// TIA Portal project "ap1_2019" (V15.1)

(* hardware
DEVICE "S7300/ET200M station_1"  S7-300 station
   slot 0: "Rail_0"  Rail  6ES7 390-1***0-0AA0
   slot 2: "PLC_1"  CPU 314C-2 PN/DP  6ES7 314-6EH04-0AB0  V3.3
      slot 2: "PROFINET interface_1"  PN-IO
         slot 1: "Port_1"  Port
         slot 2: "Port_2"  Port
      slot 5: "DI 24/DO 16_1"  DI24/DO16
      slot 6: "AI 5/AO 2_1"  AI5/AO2
      slot 7: "Count_1"  Counter
      slot 8: "Positioning_1"  Positioning
   slot 4: "DO 8x24VDC/2A_1"  DO8 x 24VDC / 2A  6ES7 322-1BF01-0AA0
DEVICE "HMI_1"  KTP900 Basic PN
   slot 0: "HMI_1"  KTP900 Basic PN  6AV2 123-2JB03-0AX0  15.1.0.0
   slot 1: "HMI_RT_1"  KTP900 Basic PN  6AV2 123-2JB03-0AX0  15.1.0.0
   slot 5: "HMI_1.IE_CP_1"  PROFINET Interface  15.0.1.0
      slot 1: "PROFINET Interface_1"  PROFINET Interface
         slot 1: "Port_1"  Port
*)

// ===== PLC "PLC_1"  CPU 314C-2 PN/DP =====

VAR_GLOBAL   // PLC tag table "Default tag table"
   "F5" AT %I0.0 : Bool;
   "S3" AT %I0.1 : Bool;
   "S4" AT %I0.2 : Bool;
   "S5" AT %I0.3 : Bool;
   "S6" AT %I0.4 : Bool;
   "S7" AT %I0.5 : Bool;
   "S8" AT %I0.6 : Bool;
   "S9" AT %I0.7 : Bool;
   "S10" AT %I1.0 : Bool;
   "S11" AT %I1.1 : Bool;
   "Reserve1" AT %I1.2 : Bool;
   "BP1" AT %I1.3 : Bool;
   "B1" AT %I1.4 : Bool;
   "B2" AT %I1.5 : Bool;
   "Reserve2" AT %I1.6 : Bool;
   "B11" AT %I1.7 : Bool;
   "B12" AT %I2.0 : Bool;
   "B21" AT %I2.1 : Bool;
   "B22" AT %I2.2 : Bool;
   "B31" AT %I2.3 : Bool;
   "B32" AT %I2.4 : Bool;
   "Reserve3" AT %I2.5 : Bool;
   "Reserve4" AT %I2.6 : Bool;
   "Reserve5" AT %I2.7 : Bool;
   "M11" AT %Q0.0 : Bool;
   "M21" AT %Q0.2 : Bool;
   "M22" AT %Q0.3 : Bool;
   "M31" AT %Q0.4 : Bool;
   "M32" AT %Q0.5 : Bool;
   "Reserve6" AT %Q0.6 : Bool;
   "Reserve7" AT %Q0.7 : Bool;
   "P32" AT %Q1.0 : Bool;
   "P33" AT %Q1.1 : Bool;
   "Reserve8" AT %Q1.2 : Bool;
   "P2" AT %Q1.3 : Bool;
   "P3" AT %Q1.4 : Bool;
   "P4" AT %Q1.5 : Bool;
   "P5" AT %Q1.6 : Bool;
   "P6" AT %Q1.7 : Bool;
   "P7" AT %Q2.0 : Bool;
   "Reserve9" AT %Q2.1 : Bool;
   "P10" AT %Q2.2 : Bool;
   "P11" AT %Q2.3 : Bool;
   "P12" AT %Q2.4 : Bool;
   "P13" AT %Q2.5 : Bool;
   "P14" AT %Q2.6 : Bool;
   "P15" AT %Q2.7 : Bool;
   "M12" AT %Q0.1 : Bool;
   "MBP1" AT %M0.0 : Bool;
   "MS3" AT %M0.1 : Bool;
   "MS4" AT %M0.2 : Bool;
   "MF5" AT %M0.3 : Bool;
   "MS5" AT %M0.4 : Bool;
   "MS6" AT %M0.5 : Bool;
   "MS7" AT %M0.6 : Bool;
   "MS8" AT %M0.7 : Bool;
   "MS9" AT %M1.0 : Bool;
   "MS10" AT %M1.1 : Bool;
   "MS11" AT %M1.2 : Bool;
   "MB1" AT %M1.3 : Bool;
   "MB2" AT %M1.4 : Bool;
END_VAR

DATA_BLOCK "Master_DB"   // DB1
{ S7_Optimized_Access := 'FALSE' }
VERSION : 0.1
// stored: InstanceOfName Master
"Master"
BEGIN
END_DATA_BLOCK

DATA_BLOCK "safety_DB"   // DB2
{ S7_Optimized_Access := 'FALSE' }
VERSION : 0.1
// stored: InstanceOfName safety
"safety"
BEGIN
END_DATA_BLOCK

DATA_BLOCK "Clock_DB"   // DB5
{ S7_Optimized_Access := 'FALSE' }
VERSION : 0.1
// stored: InstanceOfName Clock
"Clock"
BEGIN
END_DATA_BLOCK

DATA_BLOCK "Indicator_DB"   // DB6
{ S7_Optimized_Access := 'FALSE' }
VERSION : 0.1
// stored: InstanceOfName Indicator
"Indicator"
BEGIN
END_DATA_BLOCK

DATA_BLOCK "Trigger_DB"   // DB7
{ S7_Optimized_Access := 'FALSE' }
VERSION : 0.1
// stored: InstanceOfName Trigger
"Trigger"
BEGIN
END_DATA_BLOCK

DATA_BLOCK "Auto_DB"   // DB9
{ S7_Optimized_Access := 'FALSE' }
VERSION : 0.1
// stored: InstanceOfName Auto
"Auto"
BEGIN
END_DATA_BLOCK

DATA_BLOCK "HMI"   // DB14
{ S7_Optimized_Access := 'FALSE' }
VERSION : 0.1
   VAR
      "Control Panel" : Bool;
   END_VAR
BEGIN
END_DATA_BLOCK

DATA_BLOCK "Total_DB"   // DB23
{ S7_Optimized_Access := 'FALSE' }
VERSION : 0.1
// stored: InstanceOfName Total
"Total"
BEGIN
END_DATA_BLOCK

FUNCTION_BLOCK "Master"   // FB1, FBD
{ S7_Optimized_Access := 'FALSE' }
VERSION : 0.1
   VAR_INPUT
      Activate : Bool;
      BP1 : Bool;
      S3 : Bool;
      S4 : Bool;
      F5 : Bool;
   END_VAR
   VAR_OUTPUT
      G_stream : Bool;
      Operation : Bool;
   END_VAR
   VAR
      X1 : Bool;
      X2 : Bool;
      X3 : Bool;
      X4 : Bool;
      X5 : Bool;
      trick : Bool;
   END_VAR
   VAR_TEMP   // added for the SCL form of the ladder/FBD networks
      _w1 : Bool;
   END_VAR
BEGIN

REGION Network 1
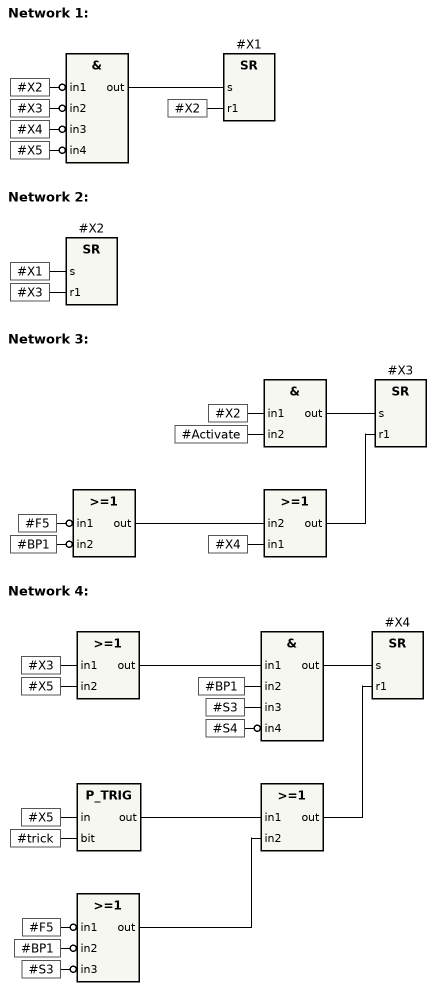
   IF NOT #X2 AND NOT #X3 AND NOT #X4 AND NOT #X5 THEN
       #X1 := TRUE;   // SR flip-flop
   END_IF;
   IF #X2 THEN #X1 := FALSE; END_IF;
END_REGION

REGION Network 2
   IF #X1 THEN
       #X2 := TRUE;   // SR flip-flop
   END_IF;
   IF #X3 THEN #X2 := FALSE; END_IF;
END_REGION

REGION Network 3
   IF #X2 AND #Activate THEN
       #X3 := TRUE;   // SR flip-flop
   END_IF;
   IF NOT #F5 OR NOT #BP1 OR #X4 THEN #X3 := FALSE; END_IF;
END_REGION

REGION Network 4
   #_w1 := #X5 AND NOT #trick;   // rising edge
   #trick := #X5;
   IF (#X3 OR #X5) AND #BP1 AND #S3 AND NOT #S4 THEN
       #X4 := TRUE;   // SR flip-flop
   END_IF;
   IF #_w1 OR NOT #F5 OR NOT #BP1 OR NOT #S3 THEN #X4 := FALSE; END_IF;
END_REGION

REGION Network 5
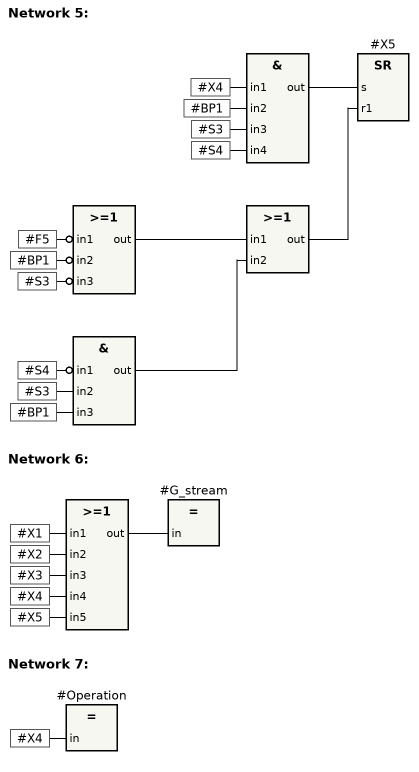
   IF #X4 AND #BP1 AND #S3 AND #S4 THEN
       #X5 := TRUE;   // SR flip-flop
   END_IF;
   IF NOT #F5 OR NOT #BP1 OR NOT #S3 OR (NOT #S4 AND #S3 AND #BP1) THEN #X5 := FALSE; END_IF;
END_REGION

REGION Network 6
   #G_stream := #X1 OR #X2 OR #X3 OR #X4 OR #X5;
END_REGION

REGION Network 7
   #Operation := #X4;
END_REGION
END_FUNCTION_BLOCK

FUNCTION_BLOCK "safety"   // FB2, FBD
{ S7_Optimized_Access := 'FALSE' }
VERSION : 0.1
   VAR_INPUT
      "G_Master.X2" : Bool;
      F5 : Bool;
      S3 : Bool;
      S4 : Bool;
      S5 : Bool;
      S6 : Bool;
      S7 : Bool;
      S8 : Bool;
      S9 : Bool;
      S10 : Bool;
      S11 : Bool;
   END_VAR
   VAR_OUTPUT
      Activate : Bool;
   END_VAR
   VAR
      X50 : Bool;
      X51 : Bool;
   END_VAR
BEGIN

REGION Network 1
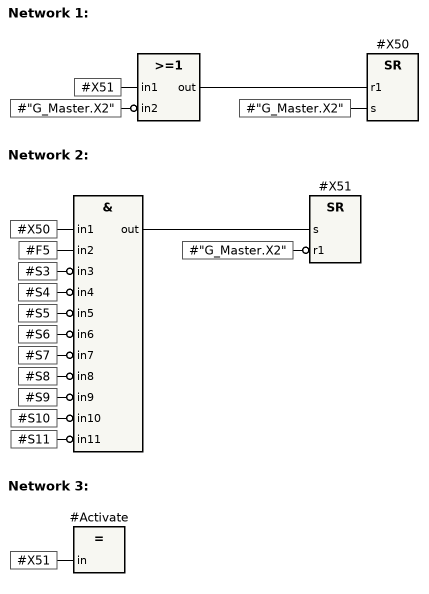
   IF #"G_Master.X2" THEN
       #X50 := TRUE;   // SR flip-flop
   END_IF;
   IF #X51 OR NOT #"G_Master.X2" THEN #X50 := FALSE; END_IF;
END_REGION

REGION Network 2
   IF #X50 AND #F5 AND NOT #S3 AND NOT #S4 AND NOT #S5 AND NOT #S6 AND NOT #S7 AND NOT #S8 AND NOT #S9 AND NOT #S10 AND NOT #S11 THEN
       #X51 := TRUE;   // SR flip-flop
   END_IF;
   IF NOT #"G_Master.X2" THEN #X51 := FALSE; END_IF;
END_REGION

REGION Network 3
   #Activate := #X51;
END_REGION
END_FUNCTION_BLOCK

FUNCTION_BLOCK "Clock"   // FB3, FBD
{ S7_Optimized_Access := 'FALSE' }
VERSION : 0.1
   VAR_OUTPUT
      "1Hz" : Bool;
   END_VAR
   VAR
      X200 : Bool;
      X201 : Bool;
   END_VAR
BEGIN

REGION Network 1
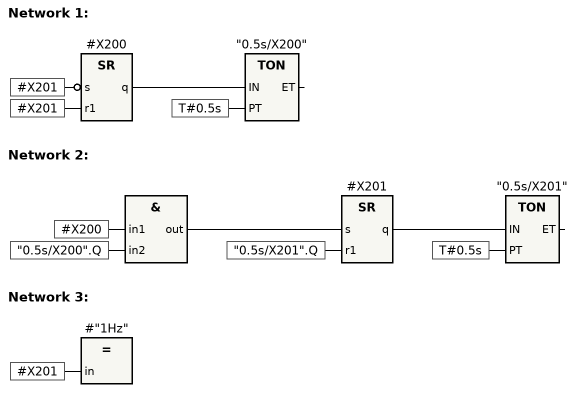
   IF NOT #X201 THEN
       #X200 := TRUE;   // SR flip-flop
   END_IF;
   IF #X201 THEN #X200 := FALSE; END_IF;
   "0.5s/X200".TON(IN := #X200, PT := T#0.5s);
END_REGION

REGION Network 2
   IF #X200 AND "0.5s/X200".Q THEN
       #X201 := TRUE;   // SR flip-flop
   END_IF;
   IF "0.5s/X201".Q THEN #X201 := FALSE; END_IF;
   "0.5s/X201".TON(IN := #X201, PT := T#0.5s);
END_REGION

REGION Network 3
   #"1Hz" := #X201;
END_REGION
END_FUNCTION_BLOCK

FUNCTION_BLOCK "Indicator"   // FB4, FBD
{ S7_Optimized_Access := 'FALSE' }
VERSION : 0.1
   VAR_INPUT
      Stream : Bool;
      S3 : Bool;
      BP1 : Bool;
      B1 : Bool;
      B2 : Bool;
      B11 : Bool;
      B12 : Bool;
      B21 : Bool;
      B22 : Bool;
      B31 : Bool;
      B32 : Bool;
      "1Hz" : Bool;
      Operation : Bool;
   END_VAR
   VAR_OUTPUT
      P2 : Bool;
      P3 : Bool;
      P4 : Bool;
      P10 : Bool;
      P11 : Bool;
      P12 : Bool;
      P13 : Bool;
      P14 : Bool;
      P15 : Bool;
      P7 : Bool;
   END_VAR
   VAR
      X100 : Bool;
      X101 : Bool;
   END_VAR
BEGIN

REGION Network 1
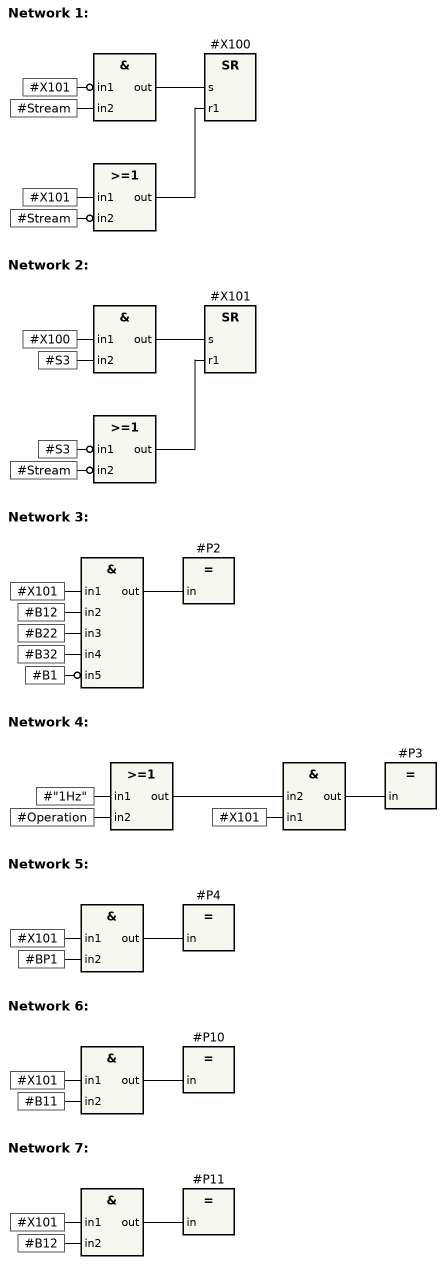
   IF NOT #X101 AND #Stream THEN
       #X100 := TRUE;   // SR flip-flop
   END_IF;
   IF #X101 OR NOT #Stream THEN #X100 := FALSE; END_IF;
END_REGION

REGION Network 2
   IF #X100 AND #S3 THEN
       #X101 := TRUE;   // SR flip-flop
   END_IF;
   IF NOT #S3 OR NOT #Stream THEN #X101 := FALSE; END_IF;
END_REGION

REGION Network 3
   #P2 := #X101 AND #B12 AND #B22 AND #B32 AND NOT #B1;
END_REGION

REGION Network 4
   #P3 := (#"1Hz" OR #Operation) AND #X101;
END_REGION

REGION Network 5
   #P4 := #X101 AND #BP1;
END_REGION

REGION Network 6
   #P10 := #X101 AND #B11;
END_REGION

REGION Network 7
   #P11 := #X101 AND #B12;
END_REGION

REGION Network 8
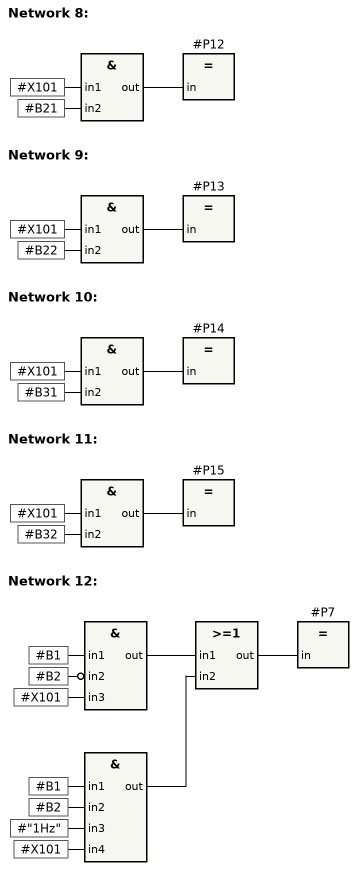
   #P12 := #X101 AND #B21;
END_REGION

REGION Network 9
   #P13 := #X101 AND #B22;
END_REGION

REGION Network 10
   #P14 := #X101 AND #B31;
END_REGION

REGION Network 11
   #P15 := #X101 AND #B32;
END_REGION

REGION Network 12
   #P7 := (#B1 AND NOT #B2 AND #X101) OR (#B1 AND #B2 AND #"1Hz" AND #X101);
END_REGION
END_FUNCTION_BLOCK

FUNCTION_BLOCK "Trigger"   // FB5, FBD
{ S7_Optimized_Access := 'FALSE' }
VERSION : 0.1
   VAR_INPUT
      "G_Master.X4" : Bool;
      S6 : Bool;
      S7 : Bool;
      S8 : Bool;
      S9 : Bool;
      S10 : Bool;
      S11 : Bool;
      B11 : Bool;
      B12 : Bool;
      B21 : Bool;
      B22 : Bool;
      B31 : Bool;
      B32 : Bool;
   END_VAR
   VAR_OUTPUT
      M11 : Bool;
      M12 : Bool;
      M21 : Bool;
      M22 : Bool;
      M31 : Bool;
      M32 : Bool;
   END_VAR
   VAR
      X20 : Bool;
   END_VAR
BEGIN

REGION Network 1
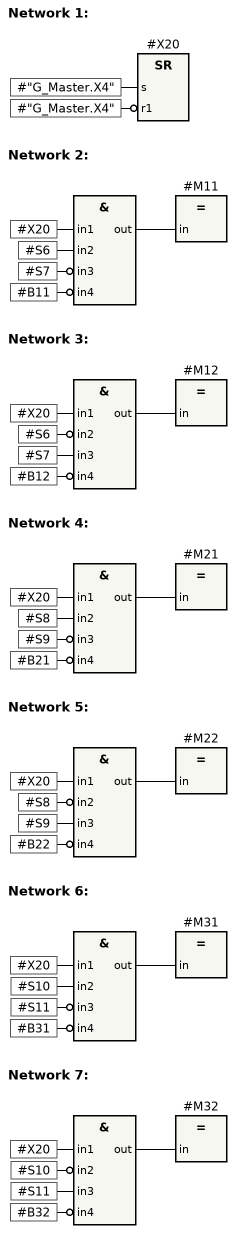
   IF #"G_Master.X4" THEN
       #X20 := TRUE;   // SR flip-flop
   END_IF;
   IF NOT #"G_Master.X4" THEN #X20 := FALSE; END_IF;
END_REGION

REGION Network 2
   #M11 := #X20 AND #S6 AND NOT #S7 AND NOT #B11;
END_REGION

REGION Network 3
   #M12 := #X20 AND NOT #S6 AND #S7 AND NOT #B12;
END_REGION

REGION Network 4
   #M21 := #X20 AND #S8 AND NOT #S9 AND NOT #B21;
END_REGION

REGION Network 5
   #M22 := #X20 AND NOT #S8 AND #S9 AND NOT #B22;
END_REGION

REGION Network 6
   #M31 := #X20 AND #S10 AND NOT #S11 AND NOT #B31;
END_REGION

REGION Network 7
   #M32 := #X20 AND NOT #S10 AND #S11 AND NOT #B32;
END_REGION
END_FUNCTION_BLOCK

FUNCTION_BLOCK "Auto"   // FB6, FBD
{ S7_Optimized_Access := 'FALSE' }
VERSION : 0.1
   VAR_INPUT
      "G_Master.X5" : Bool;
      "G_Safety.X50" : Bool;
      Operation : Bool;
      S5 : Bool;
      B1 : Bool;
      B2 : Bool;
      B11 : Bool;
      B12 : Bool;
      B21 : Bool;
      B22 : Bool;
      B31 : Bool;
      B32 : Bool;
      P2 : Bool;
   END_VAR
   VAR_OUTPUT
      M11 : Bool;
      M12 : Bool;
      M21 : Bool;
      M22 : Bool;
      M31 : Bool;
      M32 : Bool;
      P5 : Bool;
      P6 : Bool;
      P32 : Bool;
      P33 : Bool;
   END_VAR
   VAR
      X60 : Bool;
      X61 : Bool;
      X62 : Bool;
      X63 : Bool;
      X64 : Bool;
      X64a : Bool;
      X65 : Bool;
      X66 : Bool;
      X67 : Bool;
      X68 : Bool;
      X69 : Bool;
      C : Bool;
      Workpiece : Bool;
      trigger : Bool;
      Var : Int;
      MP32 : Bool;
      MP33 : Bool;
      MWP : Bool;
      MP6 : Bool;
      Quantity : DWord;
      Var_In : Int;
   END_VAR
   VAR_TEMP   // added for the SCL form of the ladder/FBD networks
      _w1 : Bool;
   END_VAR
BEGIN

REGION Network 1
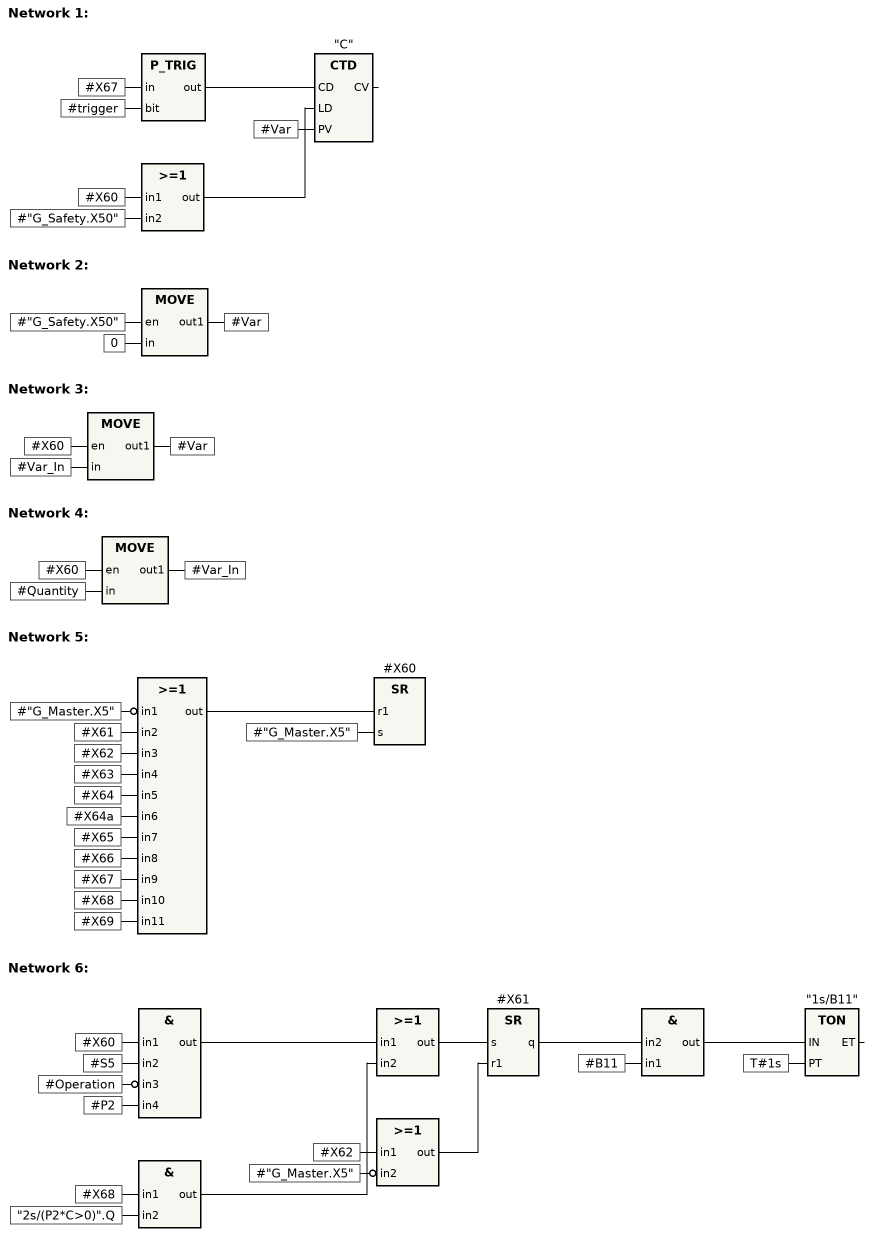
   #_w1 := #X67 AND NOT #trigger;   // rising edge
   #trigger := #X67;
   "C".CTD(CD := #_w1, LD := #X60 OR #"G_Safety.X50", PV := #Var);
END_REGION

REGION Network 2
   IF #"G_Safety.X50" THEN #Var := 0; END_IF;
END_REGION

REGION Network 3
   IF #X60 THEN #Var := #Var_In; END_IF;
END_REGION

REGION Network 4
   IF #X60 THEN #Var_In := #Quantity; END_IF;
END_REGION

REGION Network 5
   IF #"G_Master.X5" THEN
       #X60 := TRUE;   // SR flip-flop
   END_IF;
   IF NOT #"G_Master.X5" OR #X61 OR #X62 OR #X63 OR #X64 OR #X64a OR #X65 OR #X66 OR #X67 OR #X68 OR #X69 THEN
       #X60 := FALSE;
   END_IF;
END_REGION

REGION Network 6
   IF (#X60 AND #S5 AND NOT #Operation AND #P2) OR (#X68 AND "2s/(P2*C>0)".Q) THEN
       #X61 := TRUE;   // SR flip-flop
   END_IF;
   IF #X62 OR NOT #"G_Master.X5" THEN #X61 := FALSE; END_IF;
   "1s/B11".TON(IN := #X61 AND #B11, PT := T#1s);
END_REGION

REGION Network 7
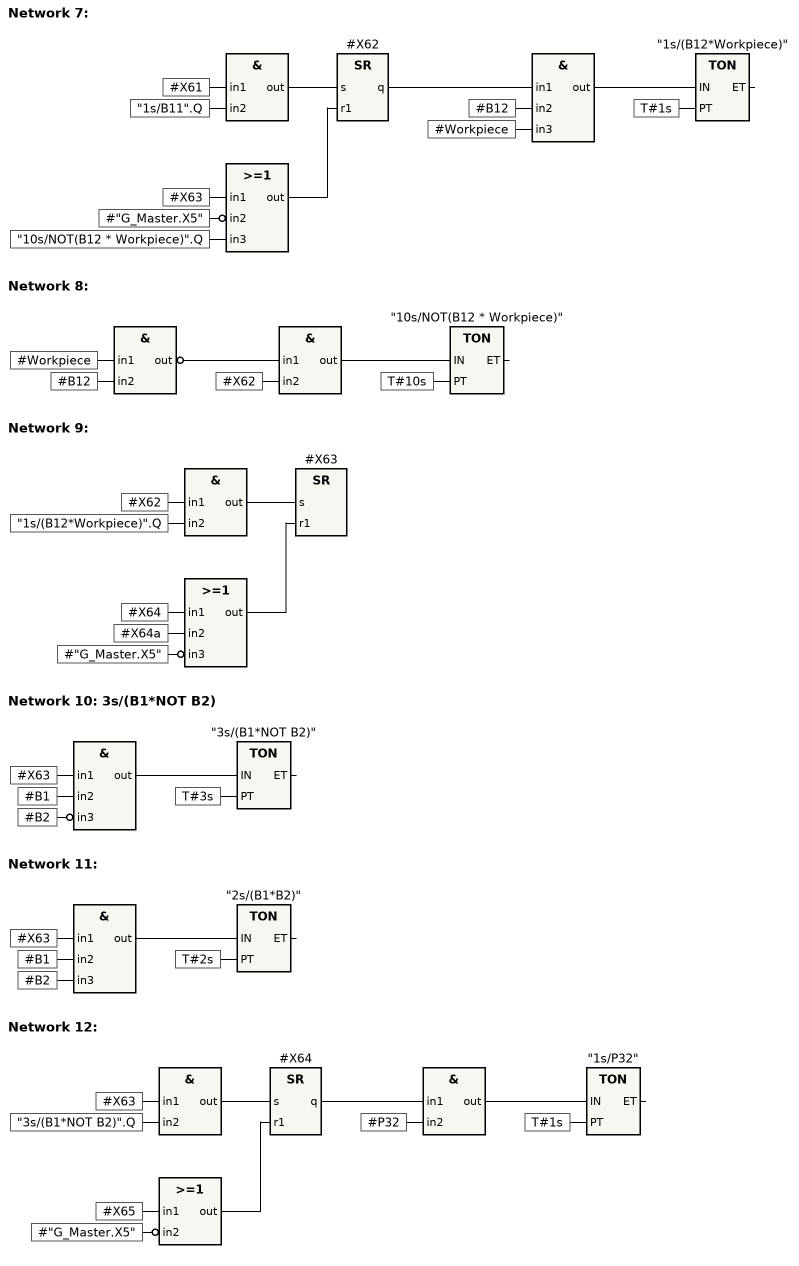
   IF #X61 AND "1s/B11".Q THEN
       #X62 := TRUE;   // SR flip-flop
   END_IF;
   IF #X63 OR NOT #"G_Master.X5" OR "10s/NOT(B12 * Workpiece)".Q THEN #X62 := FALSE; END_IF;
   "1s/(B12*Workpiece)".TON(IN := #X62 AND #B12 AND #Workpiece, PT := T#1s);
END_REGION

REGION Network 8
   "10s/NOT(B12 * Workpiece)".TON(IN := NOT (#Workpiece AND #B12) AND #X62, PT := T#10s);
END_REGION

REGION Network 9
   IF #X62 AND "1s/(B12*Workpiece)".Q THEN
       #X63 := TRUE;   // SR flip-flop
   END_IF;
   IF #X64 OR #X64a OR NOT #"G_Master.X5" THEN #X63 := FALSE; END_IF;
END_REGION

REGION Network 10: 3s/(B1*NOT B2)
   "3s/(B1*NOT B2)".TON(IN := #X63 AND #B1 AND NOT #B2, PT := T#3s);
END_REGION

REGION Network 11
   "2s/(B1*B2)".TON(IN := #X63 AND #B1 AND #B2, PT := T#2s);
END_REGION

REGION Network 12
   IF #X63 AND "3s/(B1*NOT B2)".Q THEN
       #X64 := TRUE;   // SR flip-flop
   END_IF;
   IF #X65 OR NOT #"G_Master.X5" THEN #X64 := FALSE; END_IF;
   "1s/P32".TON(IN := #X64 AND #P32, PT := T#1s);
END_REGION

REGION Network 13
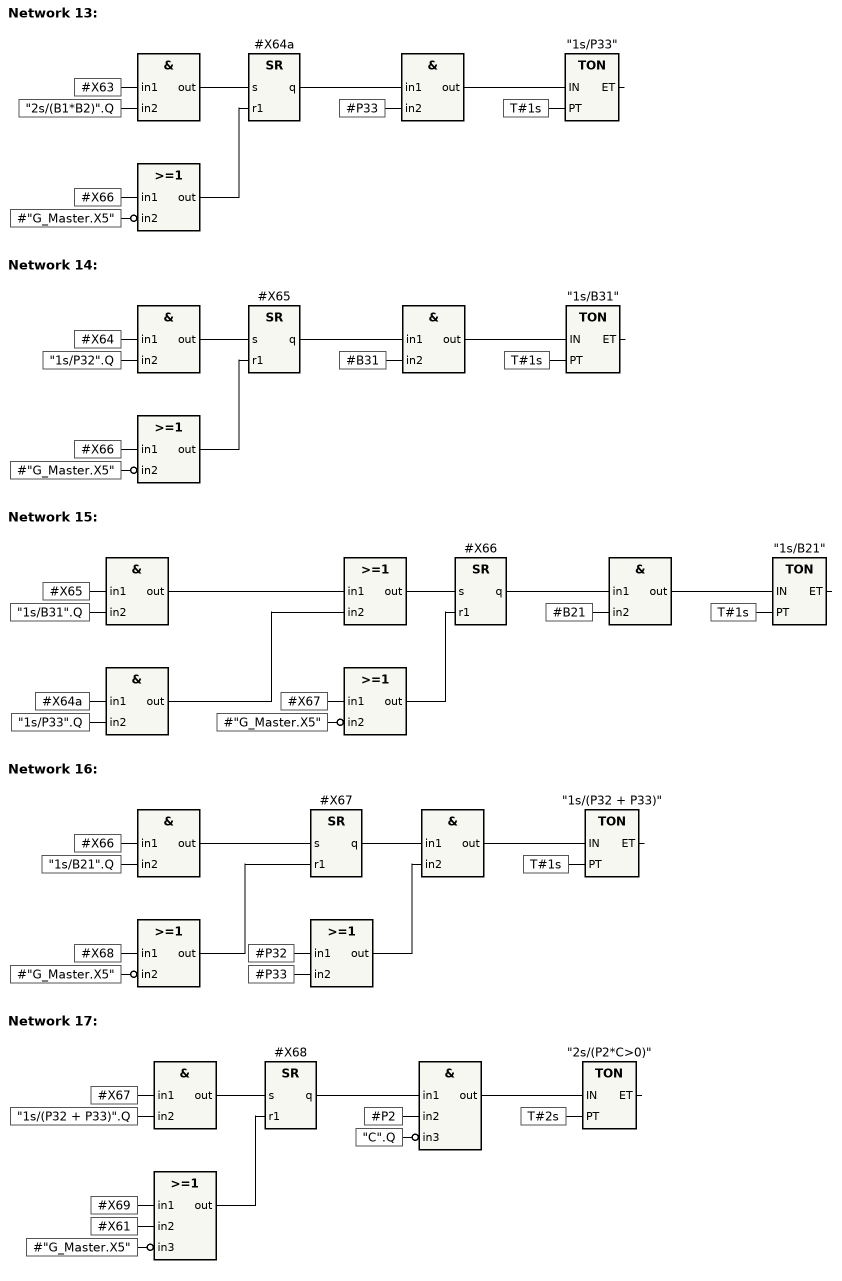
   IF #X63 AND "2s/(B1*B2)".Q THEN
       #X64a := TRUE;   // SR flip-flop
   END_IF;
   IF #X66 OR NOT #"G_Master.X5" THEN #X64a := FALSE; END_IF;
   "1s/P33".TON(IN := #X64a AND #P33, PT := T#1s);
END_REGION

REGION Network 14
   IF #X64 AND "1s/P32".Q THEN
       #X65 := TRUE;   // SR flip-flop
   END_IF;
   IF #X66 OR NOT #"G_Master.X5" THEN #X65 := FALSE; END_IF;
   "1s/B31".TON(IN := #X65 AND #B31, PT := T#1s);
END_REGION

REGION Network 15
   IF (#X65 AND "1s/B31".Q) OR (#X64a AND "1s/P33".Q) THEN
       #X66 := TRUE;   // SR flip-flop
   END_IF;
   IF #X67 OR NOT #"G_Master.X5" THEN #X66 := FALSE; END_IF;
   "1s/B21".TON(IN := #X66 AND #B21, PT := T#1s);
END_REGION

REGION Network 16
   IF #X66 AND "1s/B21".Q THEN
       #X67 := TRUE;   // SR flip-flop
   END_IF;
   IF #X68 OR NOT #"G_Master.X5" THEN #X67 := FALSE; END_IF;
   "1s/(P32 + P33)".TON(IN := #X67 AND (#P32 OR #P33), PT := T#1s);
END_REGION

REGION Network 17
   IF #X67 AND "1s/(P32 + P33)".Q THEN
       #X68 := TRUE;   // SR flip-flop
   END_IF;
   IF #X69 OR #X61 OR NOT #"G_Master.X5" THEN #X68 := FALSE; END_IF;
   "2s/(P2*C>0)".TON(IN := #X68 AND #P2 AND NOT "C".Q, PT := T#2s);
END_REGION

REGION Network 18
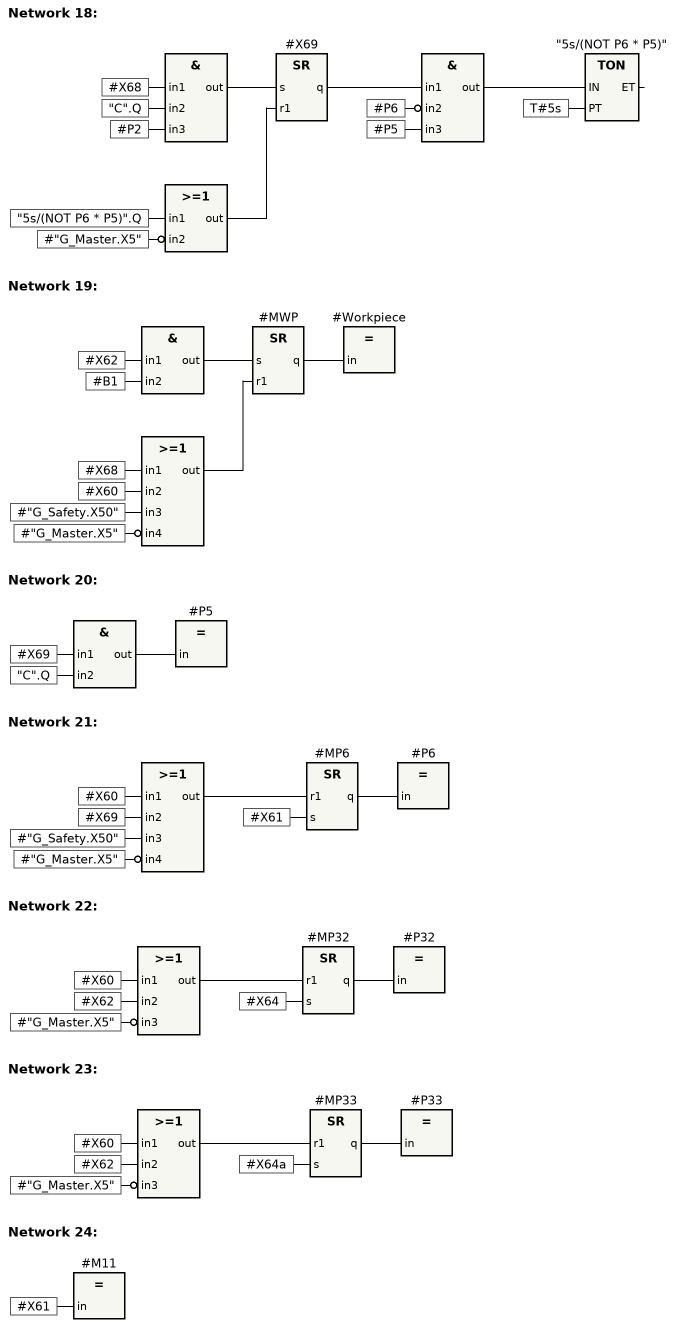
   IF #X68 AND "C".Q AND #P2 THEN
       #X69 := TRUE;   // SR flip-flop
   END_IF;
   IF "5s/(NOT P6 * P5)".Q OR NOT #"G_Master.X5" THEN #X69 := FALSE; END_IF;
   "5s/(NOT P6 * P5)".TON(IN := #X69 AND NOT #P6 AND #P5, PT := T#5s);
END_REGION

REGION Network 19
   IF #X62 AND #B1 THEN
       #MWP := TRUE;   // SR flip-flop
   END_IF;
   IF #X68 OR #X60 OR #"G_Safety.X50" OR NOT #"G_Master.X5" THEN #MWP := FALSE; END_IF;
   #Workpiece := #MWP;
END_REGION

REGION Network 20
   #P5 := #X69 AND "C".Q;
END_REGION

REGION Network 21
   IF #X61 THEN
       #MP6 := TRUE;   // SR flip-flop
   END_IF;
   IF #X60 OR #X69 OR #"G_Safety.X50" OR NOT #"G_Master.X5" THEN #MP6 := FALSE; END_IF;
   #P6 := #MP6;
END_REGION

REGION Network 22
   IF #X64 THEN
       #MP32 := TRUE;   // SR flip-flop
   END_IF;
   IF #X60 OR #X62 OR NOT #"G_Master.X5" THEN #MP32 := FALSE; END_IF;
   #P32 := #MP32;
END_REGION

REGION Network 23
   IF #X64a THEN
       #MP33 := TRUE;   // SR flip-flop
   END_IF;
   IF #X60 OR #X62 OR NOT #"G_Master.X5" THEN #MP33 := FALSE; END_IF;
   #P33 := #MP33;
END_REGION

REGION Network 24
   #M11 := #X61;
END_REGION

REGION Network 25
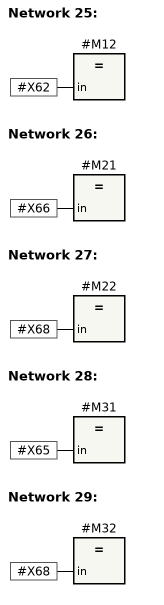
   #M12 := #X62;
END_REGION

REGION Network 26
   #M21 := #X66;
END_REGION

REGION Network 27
   #M22 := #X68;
END_REGION

REGION Network 28
   #M31 := #X65;
END_REGION

REGION Network 29
   #M32 := #X68;
END_REGION
END_FUNCTION_BLOCK

FUNCTION_BLOCK "Total"   // FB7, FBD
{ S7_Optimized_Access := 'FALSE' }
VERSION : 0.1
   VAR_INPUT
      Tgg_M11 : Bool;
      Tgg_M12 : Bool;
      Tgg_M21 : Bool;
      Tgg_M22 : Bool;
      Tgg_M31 : Bool;
      Tgg_M32 : Bool;
      Auto_M11 : Bool;
      Auto_M12 : Bool;
      Auto_M21 : Bool;
      Auto_M22 : Bool;
      Auto_M31 : Bool;
      Auto_M32 : Bool;
   END_VAR
   VAR_OUTPUT
      M11 : Bool;
      M12 : Bool;
      M21 : Bool;
      M22 : Bool;
      M31 : Bool;
      M32 : Bool;
   END_VAR
BEGIN

REGION Network 1
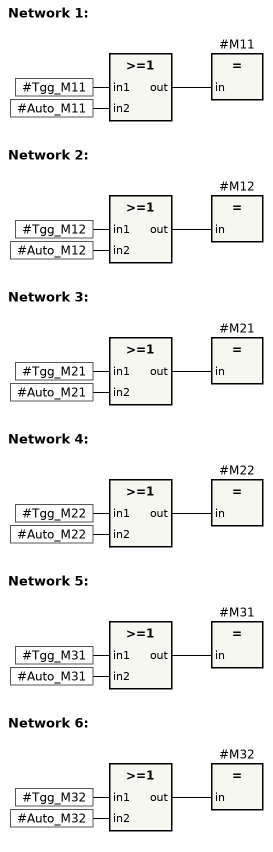
   #M11 := #Tgg_M11 OR #Auto_M11;
END_REGION

REGION Network 2
   #M12 := #Tgg_M12 OR #Auto_M12;
END_REGION

REGION Network 3
   #M21 := #Tgg_M21 OR #Auto_M21;
END_REGION

REGION Network 4
   #M22 := #Tgg_M22 OR #Auto_M22;
END_REGION

REGION Network 5
   #M31 := #Tgg_M31 OR #Auto_M31;
END_REGION

REGION Network 6
   #M32 := #Tgg_M32 OR #Auto_M32;
END_REGION
END_FUNCTION_BLOCK

ORGANIZATION_BLOCK "Main"   // OB1, FBD
TITLE = "Main Program Sweep (Cycle)"
{ S7_Optimized_Access := 'FALSE' }
VERSION : 0.1
   VAR_TEMP
      OB1_EV_CLASS : Byte;   // Bits 0-3 = 1 (Coming event), Bits 4-7 = 1 (Event class 1)
      OB1_SCAN_1 : Byte;   // 1 (Cold restart scan 1 of OB 1), 3 (Scan 2-n of OB 1)
      OB1_PRIORITY : Byte;   // Priority of OB Execution
      OB1_OB_NUMBR : Byte;   // 1 (Organization block 1, OB1)
      OB1_RESERVED_1 : Byte;   // Reserved for system
      OB1_RESERVED_2 : Byte;   // Reserved for system
      OB1_PREV_CYCLE : Int;   // Cycle time of previous OB1 scan (milliseconds)
      OB1_MIN_CYCLE : Int;   // Minimum cycle time of OB1 (milliseconds)
      OB1_MAX_CYCLE : Int;   // Maximum cycle time of OB1 (milliseconds)
      OB1_DATE_TIME : Date_And_Time;   // Date and time OB1 started
   END_VAR
BEGIN

REGION Network 1
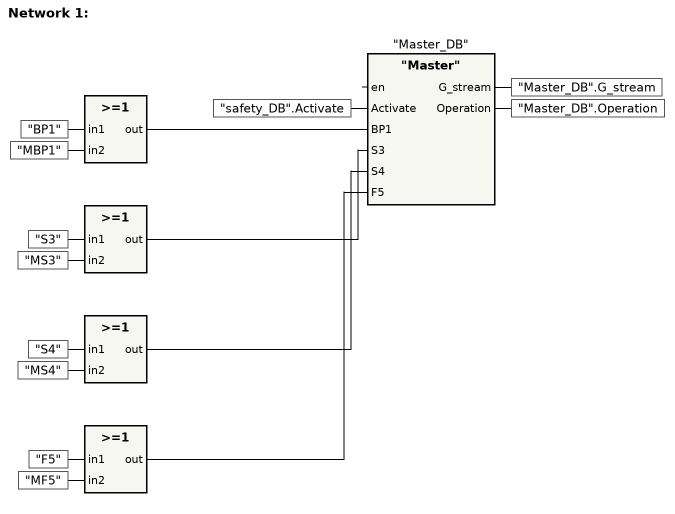
   "Master_DB"(Activate := "safety_DB".Activate,   // "Master"
               BP1 := "BP1" OR "MBP1",
               S3 := "S3" OR "MS3",
               S4 := "S4" OR "MS4",
               F5 := "F5" OR "MF5",
               G_stream => "Master_DB".G_stream,
               Operation => "Master_DB".Operation);
END_REGION

REGION Network 2
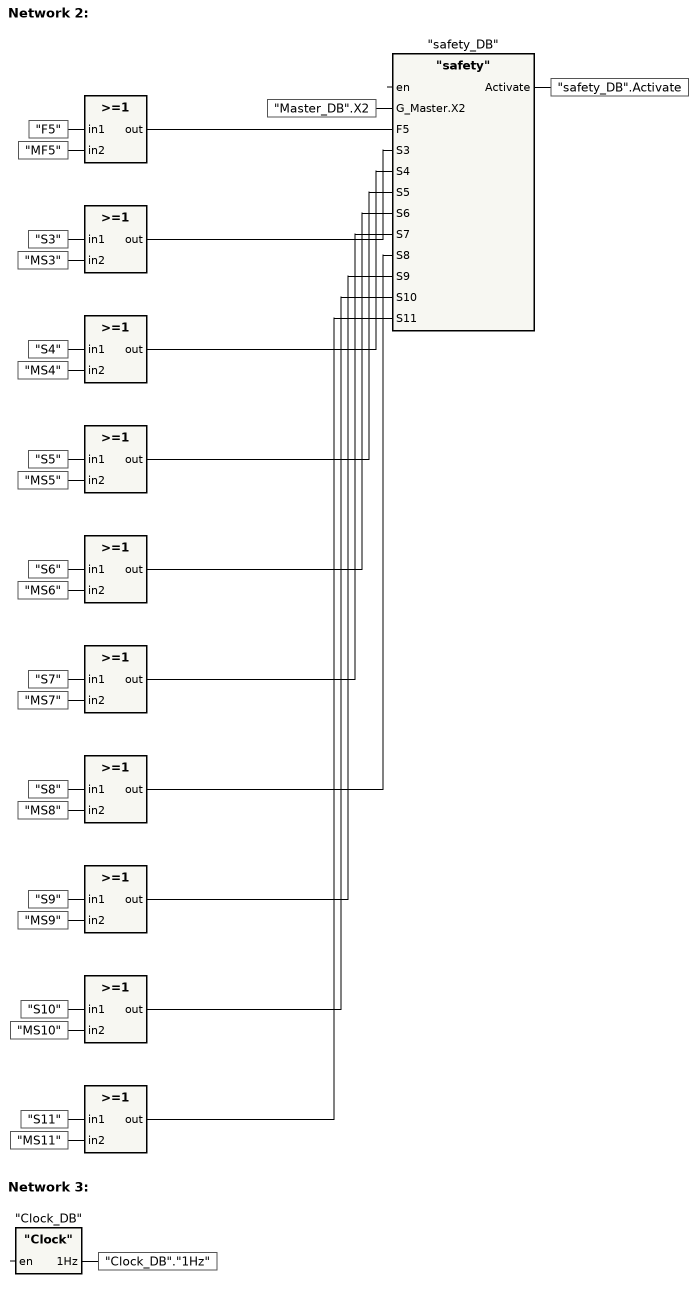
   "safety_DB"("G_Master.X2" := "Master_DB".X2,   // "safety"
               F5 := "F5" OR "MF5",
               S3 := "S3" OR "MS3",
               S4 := "S4" OR "MS4",
               S5 := "S5" OR "MS5",
               S6 := "S6" OR "MS6",
               S7 := "S7" OR "MS7",
               S8 := "S8" OR "MS8",
               S9 := "S9" OR "MS9",
               S10 := "S10" OR "MS10",
               S11 := "S11" OR "MS11",
               Activate => "safety_DB".Activate);
END_REGION

REGION Network 3
   "Clock_DB"("1Hz" => "Clock_DB"."1Hz");   // "Clock"
END_REGION

REGION Network 4
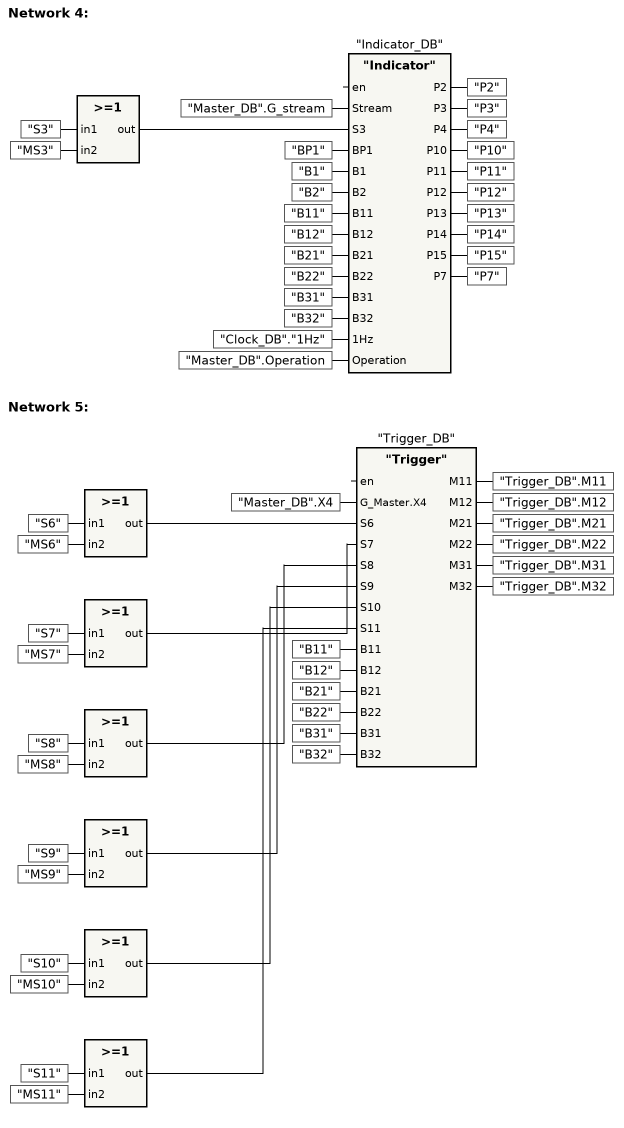
   "Indicator_DB"(Stream := "Master_DB".G_stream,   // "Indicator"
                  S3 := "S3" OR "MS3",
                  BP1 := "BP1",
                  B1 := "B1",
                  B2 := "B2",
                  B11 := "B11",
                  B12 := "B12",
                  B21 := "B21",
                  B22 := "B22",
                  B31 := "B31",
                  B32 := "B32",
                  "1Hz" := "Clock_DB"."1Hz",
                  Operation := "Master_DB".Operation,
                  P2 => "P2",
                  P3 => "P3",
                  P4 => "P4",
                  P10 => "P10",
                  P11 => "P11",
                  P12 => "P12",
                  P13 => "P13",
                  P14 => "P14",
                  P15 => "P15",
                  P7 => "P7");
END_REGION

REGION Network 5
   "Trigger_DB"("G_Master.X4" := "Master_DB".X4,   // "Trigger"
                S6 := "S6" OR "MS6",
                S7 := "S7" OR "MS7",
                S8 := "S8" OR "MS8",
                S9 := "S9" OR "MS9",
                S10 := "S10" OR "MS10",
                S11 := "S11" OR "MS11",
                B11 := "B11",
                B12 := "B12",
                B21 := "B21",
                B22 := "B22",
                B31 := "B31",
                B32 := "B32",
                M11 => "Trigger_DB".M11,
                M12 => "Trigger_DB".M12,
                M21 => "Trigger_DB".M21,
                M22 => "Trigger_DB".M22,
                M31 => "Trigger_DB".M31,
                M32 => "Trigger_DB".M32);
END_REGION

REGION Network 6
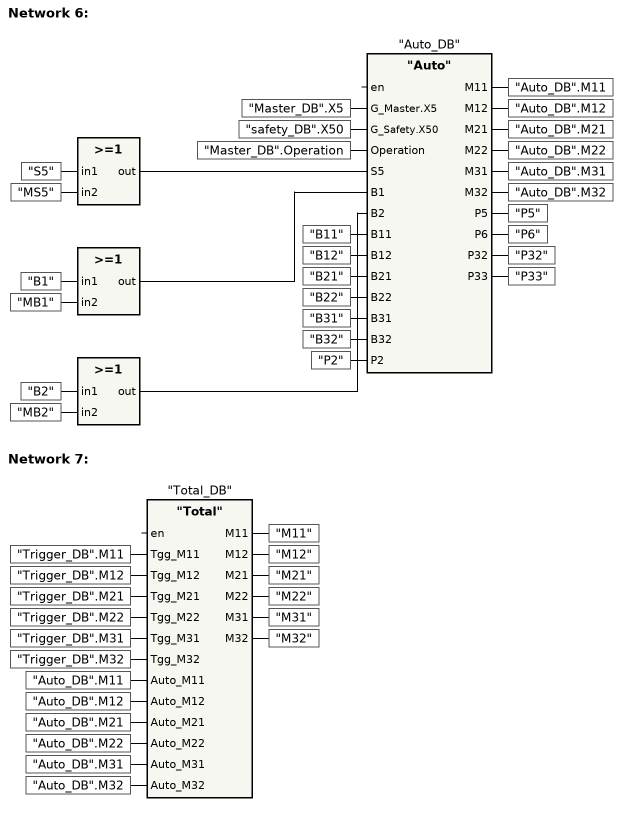
   "Auto_DB"("G_Master.X5" := "Master_DB".X5,   // "Auto"
             "G_Safety.X50" := "safety_DB".X50,
             Operation := "Master_DB".Operation,
             S5 := "S5" OR "MS5",
             B1 := "B1" OR "MB1",
             B2 := "B2" OR "MB2",
             B11 := "B11",
             B12 := "B12",
             B21 := "B21",
             B22 := "B22",
             B31 := "B31",
             B32 := "B32",
             P2 := "P2",
             M11 => "Auto_DB".M11,
             M12 => "Auto_DB".M12,
             M21 => "Auto_DB".M21,
             M22 => "Auto_DB".M22,
             M31 => "Auto_DB".M31,
             M32 => "Auto_DB".M32,
             P5 => "P5",
             P6 => "P6",
             P32 => "P32",
             P33 => "P33");
END_REGION

REGION Network 7
   "Total_DB"(Tgg_M11 := "Trigger_DB".M11,   // "Total"
              Tgg_M12 := "Trigger_DB".M12,
              Tgg_M21 := "Trigger_DB".M21,
              Tgg_M22 := "Trigger_DB".M22,
              Tgg_M31 := "Trigger_DB".M31,
              Tgg_M32 := "Trigger_DB".M32,
              Auto_M11 := "Auto_DB".M11,
              Auto_M12 := "Auto_DB".M12,
              Auto_M21 := "Auto_DB".M21,
              Auto_M22 := "Auto_DB".M22,
              Auto_M31 := "Auto_DB".M31,
              Auto_M32 := "Auto_DB".M32,
              M11 => "M11",
              M12 => "M12",
              M21 => "M21",
              M22 => "M22",
              M31 => "M31",
              M32 => "M32");
END_REGION
END_ORGANIZATION_BLOCK

(* ===== HMI "HMI_RT_1" =====
system functions are stored by id; their names below are inferred from use
connection "HMI_Connection_1": ETHERNET, SIMATIC S7 300/400 MPI

HMI tags "Default tag table"
   "Tag_ScreenNumber" : UInt, internal
   "HMI_Control Panel" : Bool, internal
   "MF5" : Bool = PLC MF5 AT %M0.3, 100 ms
   "Indicator_DB_P3" : Bool = PLC Indicator_DB.P3 AT %DB6.DBX2.1, 100 ms
   "Indicator_DB_P2" : Bool = PLC Indicator_DB.P2 AT %DB6.DBX2.0, 100 ms
   "MS3" : Bool = PLC MS3 AT %M0.1, 100 ms
   "P3" : Bool = PLC P3 AT %Q1.4, 100 ms
   "MS4" : Bool = PLC MS4 AT %M0.2, 100 ms
   "MS5" : Bool = PLC MS5 AT %M0.4, 100 ms
   "MS6" : Bool = PLC MS6 AT %M0.5, 100 ms
   "MS7" : Bool = PLC MS7 AT %M0.6, 100 ms
   "P4" : Bool = PLC P4 AT %Q1.5, 100 ms
   "P2" : Bool = PLC P2 AT %Q1.3, 100 ms
   "P7" : Bool = PLC P7 AT %Q2.0, 100 ms
   "MS8" : Bool = PLC MS8 AT %M0.7, 100 ms
   "MS9" : Bool = PLC MS9 AT %M1.0, 100 ms
   "MS10" : Bool = PLC MS10 AT %M1.1, 100 ms
   "MS11" : Bool = PLC MS11 AT %M1.2, 100 ms
   "MB1" : Bool = PLC MB1 AT %M1.3, 100 ms
   "P10" : Bool = PLC P10 AT %Q2.2, 100 ms
   "P11" : Bool = PLC P11 AT %Q2.3, 100 ms
   "P12" : Bool = PLC P12 AT %Q2.4, 100 ms
   "P13" : Bool = PLC P13 AT %Q2.5, 100 ms
   "P14" : Bool = PLC P14 AT %Q2.6, 100 ms
   "P15" : Bool = PLC P15 AT %Q2.7, 100 ms
   "P5" : Bool = PLC P5 AT %Q1.6, 100 ms
   "P6" : Bool = PLC P6 AT %Q1.7, 100 ms
   "Root" : Bool, internal
   "Process" : Bool, internal
   "F5" : Bool = PLC F5 AT %I0.0, 100 ms
   "BP1" : Bool = PLC BP1 AT %I1.3, 100 ms
   "MB2" : Bool = PLC MB2 AT %M1.4, 1 s
   "Master_DB_F5" : Bool = PLC Master_DB.F5 AT %DB1.DBX0.4, 1 s
   "Auto_DB_MP6" : Bool = PLC Auto_DB.MP6 AT %DB9.DBX8.3, 1 s
   "Auto_DB_Quantity" : DWord = PLC Auto_DB.Quantity AT %DB9.DBD10, 1 s
   "Indicator_DB_B1" : Bool = PLC Indicator_DB.B1 AT %DB6.DBX0.3, 1 s
   "Indicator_DB_B2" : Bool = PLC Indicator_DB.B2 AT %DB6.DBX0.4, 1 s

graphic list "@DiagnosticsStates": 0 '@Diagnostics_StateGood'; 1 '@Diagnostics_StateBad'

Template "Template_1" 800x480
   Button "Exit" at 722,440 size 55x39; TextOff 'Exit'; PictureOff "ExitRuntime_KTP900_Basic_PN_TR"; PictureOn "ExitRuntime_KTP900_Basic_PN_TR"
      on Release: StopRuntime(0)
   Button "Template_Button" at 622,440 size 55x39; TextOff 'Text'
   Button "Template_Button_1" at 522,440 size 55x39; TextOff 'Text'
   Button "Template_Button_2" at 422,440 size 55x39; TextOff 'Text'
   Button "Template_Button_3" at 322,440 size 55x39; TextOff 'Text'
   Button "Template_Button_4" at 222,440 size 55x39; TextOff 'Text'
   Button "Alarms" at 122,440 size 55x39; TextOff 'Alarms'; PictureOff "AlarmDisplay_KTP900_Basic_PN_TR"; PictureOn "AlarmDisplay_KTP900_Basic_PN_TR"
      on Release: function_ef3f5d25("Alarm window_Unacknowledged", -1)
   Button "Start screen" at 22,440 size 55x39; TextOff 'Start screen'; PictureOff "NavigateHome_KTP900_Basic_PN_TR"; PictureOn "NavigateHome_KTP900_Basic_PN_TR"
      on Release: ActivateScreen("Root screen", 0)
   SymbolicIOField "Symbolic_IO_Field_Screen" at 73,7 size 620x26; TextOff '0'; TextOn '1'; TextList "TextList_ScreenNames"
      ProcessValue <- "Tag_ScreenNumber"
      on Change: ActivateScreenByNumber("Tag_ScreenNumber", 0)
   DateTimeField "HmiScreenItemData" at 695,20 size 105x20
   DateTimeField "HmiScreenItemData_1" at 695,0 size 105x20
   GraphicView "Logo" at 0,0 size 71x40; Picture "Logo of HMI_1"

screen "Root screen" 800x480, template "Template_1"
   on GenerateScreen: SetTag("Tag_ScreenNumber", 1)
   GraphicView "Graphic view_1" at 417,132 size 358x298; Picture "OIP"
   Button "Button_1" at 42,355 size 137x51; TextOff 'Control Panel'
      Appearance <- "HMI_Control Panel"
      on Press: SetBit("HMI_Control Panel"); ActivateScreen("Control", 0)
      on Release: ResetBit("HMI_Control Panel")
   GraphicView "Graphic view_2" at 261,211 size 141x111; Picture "Graphic_3"
   GraphicView "Graphic view_3" at 42,206 size 140x142; Picture "Graphic_4"
   Button "Button_2" at 268,355 size 137x51; TextOff 'Process'
      on Release: ResetBit("HMI_Control Panel")
      on Press: SetBit("Process"); ActivateScreen("Process", 0)
      Appearance <- "HMI_Control Panel"

screen "Control" 800x480
   Switch "Pushbutton_Emergency" at 34,16 size 80x80; CaptionText 'Switch'; TextOff '0'; TextOn '1'; PictureOff "Pushbutton_Emergency_Off_256c"; PictureOn "Pushbutton_Emergency_On_256c"
      on SwitchOn: ResetBit("Master_DB_F5")
      on SwitchOff: SetBit("Master_DB_F5")
   Switch "Rotary_N_Mono" at 34,309 size 80x80; CaptionText 'Switch'; TextOff '0'; TextOn '1'; PictureOff "Rotary_N_Off_mono"; PictureOn "Rotary_N_On_mono"
      on SwitchOn: SetBit("MS3")
      on SwitchOff: ResetBit("MS3")
   Switch "Rotary_N_Mono_1" at 176,164 size 80x80; CaptionText 'Switch'; TextOff '0'; TextOn '1'; PictureOff "Rotary_N_Off_mono"; PictureOn "Rotary_N_On_mono"
      on SwitchOn: SetBit("MS4")
      on SwitchOff: ResetBit("MS4")
   Button "FB_Empty_Round" at 34,164 size 86x89; TextOff 'Text'; PictureOn "FB_Empty_Round_Pressed_256c"; PictureOff "Pushbutton_Round_N_On_mono"
      on Press: ResetBit("Master_DB_F5")
      on Release: SetBit("Master_DB_F5")
      Appearance <- "MF5"
   Button "FB_Empty_Round_1" at 303,13 size 86x89; TextOff 'Text'; PictureOn "FB_Empty_Round_Pressed_256c"; PictureOff "Pushbutton_Round_N_On_mono"
      on Press: SetBit("MS6")
      on Release: ResetBit("MS6")
   Button "FB_Empty_Round_2" at 444,13 size 86x89; TextOff 'Text'; PictureOn "FB_Empty_Round_Pressed_256c"; PictureOff "Pushbutton_Round_N_On_mono"
      on Press: SetBit("MS7")
      on Release: ResetBit("MS7")
   Button "FB_Empty_Round_3" at 303,161 size 86x89; TextOff 'Text'; PictureOn "FB_Empty_Round_Pressed_256c"; PictureOff "Pushbutton_Round_N_On_mono"
      on Press: SetBit("MS8")
      on Release: ResetBit("MS8")
   Button "FB_Empty_Round_4" at 444,161 size 86x89; TextOff 'Text'; PictureOn "FB_Empty_Round_Pressed_256c"; PictureOff "Pushbutton_Round_N_On_mono"
      on Release: ResetBit("MS9")
      on Press: SetBit("MS9")
   Button "FB_Empty_Round_5" at 303,306 size 86x89; TextOff 'Text'; PictureOn "FB_Empty_Round_Pressed_256c"; PictureOff "Pushbutton_Round_N_On_mono"
      on Press: SetBit("MS10")
      on Release: ResetBit("MS10")
   Button "FB_Empty_Round_6" at 444,306 size 86x89; TextOff 'Text'; PictureOn "FB_Empty_Round_Pressed_256c"; PictureOff "Pushbutton_Round_N_On_mono"
      on Press: SetBit("MS11")
      on Release: ResetBit("MS11")
   Button "FB_Empty_Round_7" at 171,306 size 86x89; TextOff 'Text'; PictureOn "FB_Empty_Round_Pressed_256c"; PictureOff "Pushbutton_Round_N_On_mono"
      on Press: SetBit("MS5")
      on Release: ResetBit("MS5")
   Circle "Circle_2" at 43,174 size 67x67
      Visibility <- "Master_DB_F5"
   Circle "Circle_3" at 312,23 size 67x67
      Visibility <- "P10"
   Circle "Circle_4" at 453,23 size 67x67
      Visibility <- "P11"
   Circle "Circle_5" at 312,171 size 67x67
      Visibility <- "P12"
   Circle "Circle_6" at 453,171 size 67x67
      Visibility <- "P13"
   Circle "Circle_7" at 312,316 size 67x67
      Visibility <- "P14"
   Circle "Circle_8" at 453,316 size 67x67
      Visibility <- "P15"
   Circle "Circle_1" at 176,20 size 74x74
      Appearance <- "P3"
   Circle "Circle_9" at 577,20 size 74x74
      Appearance <- "P7"
   Circle "Circle_10" at 699,20 size 74x74
      Appearance <- "P4"
   Circle "Circle_11" at 699,168 size 74x74
      Appearance <- "P2"
   Circle "Circle_12" at 699,314 size 74x74
      Appearance <- "P5"
   Circle "Circle_13" at 180,316 size 67x67
      Visibility <- "P6"
   TextField "Text field_1" at 16,101 size 110x36; Text 'S1 Emergency Stop'
   TextField "Text field_2" at 16,253 size 118x36; Text 'S2 Reset Emergency'
   TextField "Text field_3" at 43,395 size 61x36; Text 'S3 Activate'
   TextField "Text field_4" at 176,397 size 81x36; Text 'S5/P6 Start/Cycle'
   TextField "Text field_5" at 170,253 size 91x36; Text 'S4 Trigger/Auto'
   TextField "Text field_6" at 172,99 size 91x36; Text 'P3 Trigger/Auto'
   TextField "Text field_7" at 304,100 size 78x36; Text 'S6/P10 M10 return'
   TextField "Text field_8" at 452,100 size 81x36; Text 'S7/P11 M10 extend'
   TextField "Text field_9" at 454,251 size 81x36; Text 'S9/13 M20 extend'
   TextField "Text field_10" at 308,252 size 78x36; Text 'S8/P12 M20 return'
   TextField "Text field_11" at 455,395 size 81x36; Text 'S11/P15 M30 extend'
   TextField "Text field_12" at 309,395 size 78x36; Text 'S10/P14 M30 return'
   TextField "Text field_13" at 581,99 size 70x36; Text 'P7 Billes/Slot'
   TextField "Text field_14" at 678,97 size 114x36; Text 'P4 Enough pressure'
   TextField "Text field_15" at 688,251 size 96x36; Text 'P2 Initial position'
   TextField "Text field_16" at 708,392 size 61x36; Text 'P5 Quantity'
   Button "Button_1" at 688,441 size 108x38; TextOff 'Home'
      on Release: ResetBit("HMI_Control Panel")
      on Press: SetBit("Root"); ActivateScreen("Root screen", 0)
      Appearance <- "HMI_Control Panel"
   Button "Button_2" at 552,441 size 108x38; TextOff 'Process'
      on Release: ResetBit("HMI_Control Panel")
      on Press: SetBit("Process"); ActivateScreen("Process", 0)
      Appearance <- "HMI_Control Panel"
   Switch "Switch_1" at 50,443 size 64x32; CaptionText 'Switch'; TextOff 'OFF'; TextOn 'ON'
      on SwitchOn: SetBit("MB1")
      on SwitchOff: ResetBit("MB1")
   Switch "Switch_2" at 184,444 size 64x32; TextOn 'ON'; CaptionText 'Switch'; TextOff 'OFF'
      on SwitchOff: ResetBit("MB2")
      on SwitchOn: SetBit("MB2")
   TextField "Text field_17" at 23,453 size 21x20; Text 'B1'
   TextField "Text field_18" at 156,453 size 21x20; Text 'B2'
   IOField "I/O field_1" at 263,445 size 96x32; FormatPattern 999
      ProcessValue <- "Auto_DB_Quantity"

screen "Process" 800x480
   Button "Button_1" at 688,441 size 108x38; TextOff 'Home'
      on Release: ResetBit("HMI_Control Panel")
      on Press: SetBit("Root"); ActivateScreen("Root screen", 0)
      Appearance <- "HMI_Control Panel"
   Button "Button_2" at 552,441 size 108x38; TextOff 'Control Panel'
      on Release: ResetBit("HMI_Control Panel")
      on Press: SetBit("HMI_Control Panel"); ActivateScreen("Control", 0)
      Appearance <- "HMI_Control Panel"
*)